{attribute 'qualified_only'}
{attribute 'strict'}
TYPE Enum_Presence :
(
	Non_presence := 0,				
	Presence
);
END_TYPE

(* stored: Version 1.1.0.1, ProductVersion 3.1.4022.18
   DUT Enum_Presence: Id {fe94b97e-5a51-49cf-a0c2-585b97c6fe9b} *)
